(* CODESYS project Ladder v1_RECOVERED_2026-06-05T00-47-06.project

Project tree, tasks and I/O mapping:
  Device : CODESYS Control Win V3 x64, CODESYS, version 3.5.21.30
    application Application
      libraries: Standard, 3.5.18.0 (System)
      task MainTask (cyclic, interval t#20ms, priority 1) calls PLC_PRG
      Symbols
      program PLC_PRG [LD]
      Symbols
*)

// Device/Application/PLC_PRG
PROGRAM PLC_PRG
VAR
    ///////////////////////////
    // PLC Inputs / Factory I/O Sensors
    ///////////////////////////

    IN_Moving_X_Sensor        : BOOL; // Moving X
    IN_Moving_Z_Sensor        : BOOL; // Moving Z
    IN_Item_Detected          : BOOL; // Item detected
    IN_Lid_At_Place           : BOOL; // Lid at place
    IN_Lid_Clamped            : BOOL; // Lid clamped
    IN_Lid_Pos_At_Limit       : BOOL; // Pos. at limit lids
    IN_Base_At_Place          : BOOL; // Base at place
    IN_Base_Clamped           : BOOL; // Base clamped
    IN_Base_Pos_At_Limit      : BOOL; // Pos. at limit bases
    IN_Part_Leaving           : BOOL; // Part leaving

    IN_Start                  : BOOL; // Start button
    IN_Reset                  : BOOL; // Reset button
    IN_Stop                   : BOOL; // Stop button
    IN_EStop                  : BOOL; // Emergency stop
    IN_Auto_Mode              : BOOL; // Auto
    IN_FactoryIO_Running      : BOOL; // FACTORY I/O Running


    //////////////////////////////////
    // PLC Outputs / Factory I/O Actuators
    //////////////////////////////////

    OUT_Move_X                : BOOL; // Move X
    OUT_Move_Z                : BOOL; // Move Z
    OUT_Grab                  : BOOL; // Grab
    OUT_Lids_Conveyor         : BOOL; // Lids conveyor
    OUT_Clamp_Lid             : BOOL; // Clamp lid
    OUT_Raise_Lid_Position    : BOOL; // Pos. raise lids
    OUT_Bases_Conveyor        : BOOL; // Bases conveyor
    OUT_Clamp_Base            : BOOL; // Clamp base
    OUT_Raise_Base_Position   : BOOL; // Pos. raise bases

    OUT_Start_Light           : BOOL; // Start light
    OUT_Reset_Light           : BOOL; // Reset light
    OUT_Stop_Light            : BOOL; // Stop light

    OUT_Counter               : INT; // Counter


    ///////////////////////////////
    // Internal vars
    ///////////////////////////////

    M_Step_Num                : INT; // Step

	TON_0: TON;
	T0: TIME;
	CTU_0: CTU;
END_VAR
VAR // added by the converter: edge detectors and wires of the graphical bodies
    _w1 : BOOL;
END_VAR

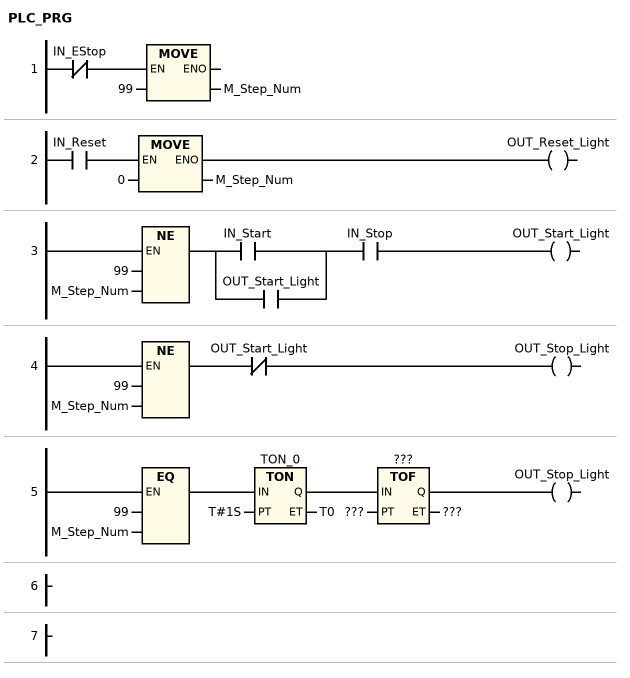
// NETWORK 1
IF NOT IN_EStop THEN M_Step_Num := 99; END_IF

// NETWORK 2
_w1 := IN_Reset;
IF _w1 THEN M_Step_Num := 0; END_IF
OUT_Reset_Light := _w1;

// NETWORK 3
OUT_Start_Light := 99 <> M_Step_Num AND (IN_Start OR OUT_Start_Light) AND IN_Stop;

// NETWORK 4
OUT_Stop_Light := 99 <> M_Step_Num AND NOT OUT_Start_Light;

// NETWORK 5
TON_0(IN := 99 = M_Step_Num, PT := T#1S, ET => T0); // TON
???(IN := TON_0.Q); // TOF
OUT_Stop_Light := ???.Q;

// NETWORK 6

// NETWORK 7

END_PROGRAM
